INTERFACE I_CyclicInstance EXTENDS __SYSTEM.IQueryInterface

PROPERTY PUBLIC CyclicInstanceCallback : I_Callback
GET
END_GET
END_PROPERTY

END_INTERFACE

(* stored: Version 1.1.0.1, ProductVersion 3.1.4024.11
   Itf I_CyclicInstance: Id {4754e690-be22-46b2-a638-e12e81147fb2}
   Property CyclicInstanceCallback: Id {b7cc4041-9e45-4cf0-9ed6-2e3d302391a8}
   Get Get: Id {2d51a4cd-e69a-4d27-9009-334dafb249fc} *)
